{attribute 'qualified_only'}
{attribute 'to_string'}
TYPE E_JointSetupStates :
(
	Idle:=0,
	SetAbsEncoderPositiveDir,
	SetAbsEncoderScale,
	SetAbsEncoderOffset,
	SetIncEncoderPositiveDir,
	SetIncEncoderScale,
	SaveAbsEncPosAndIncEncoderOffset,
	SetIncEncHome,
	WrapUp
)UINT := Idle
;
END_TYPE

(* stored: Version 1.1.0.1, ProductVersion 3.1.4024.12
   EnumerationTextList E_JointSetupStates: Id {2a6792d0-30e4-4f5e-bb11-2ac9c32a1265} *)
